INTERFACE I_MirrorCover

METHOD Close : BOOL
VAR_INPUT
END_VAR
END_METHOD

METHOD Open : BOOL
VAR_INPUT
END_VAR
END_METHOD

END_INTERFACE

(* stored: Version 1.1.0.1, ProductVersion 3.1.4024.12
   Itf I_MirrorCover: Id {ce637c3e-ed3e-4174-8b7f-5e29873c1a6c}
   Method Close: Id {d170ed42-b733-4dca-b829-4ce12e150295}
   Method Open: Id {47330435-4ab9-4214-8907-9d0910956eeb} *)
